(*			
	EVERDE sp. z o.o.
	Rafał Osajda		08.08.2025		TC 4024.66
	Interfejs do wyciągania z SPM przez HMI danych do wyświetlania - dla Ramki głównej tryb produkcja
*)
INTERFACE ITF_SPM_HMI_00_01_Lacznik EXTENDS  B_Baza.ITF_ZrodloIdentyfikacji

END_INTERFACE

(* stored: Version 1.1.0.1
   Itf ITF_SPM_HMI_00_01_Lacznik: Id {d5105468-53b8-072d-0a25-d1e3b8822896} *)
